// TwinCAT 3 PLC project PLC3
// ProgramVersion: 3.1.4022.3
// libraries:
//   Tc2_Standard, * (Beckhoff Automation GmbH)
//   Tc2_System, * (Beckhoff Automation GmbH)
//   Tc3_Module, * (Beckhoff Automation GmbH)
// project tree:
//   DUTs/ States.TcDUT (not stored)
//   / GlobalTextList.TcGTLO (not stored), PlcTask.TcTTO (not stored), Visualization Manager.TcVMO (not stored)
//   GVLs/ GVL_IO.TcGVL (not stored)
//   POUs/ MAIN.TcPOU, Moving.TcPOU
//   VISUs/ Visualization.TcVIS

// ---- POUs/MAIN.TcPOU
PROGRAM MAIN
VAR
	Timer1 :TON;
	Timer2 : TON;
	PulseTimer1 : TP;

	CurrentState  : States;
	
	ServoRTrigY : R_Trig ; 
	ServoRTrigX : R_Trig ; 
	
	//Eigen trigger booleans
	InitYReady : BOOL;
	InitXReady : BOOL;

	Test : Moving;
	Pos : INT;
	ActualPos : int;
END_VAR

PulseTimer1(IN:=GVL_IO.Start_button, PT:=T#150MS);

Timer1(IN:= GVL_IO.a_1_Vertical_Zaxis_downward, PT:= T#10MS);

CASE CurrentState OF
States.Init:
		//Aanzetten van servo's. Dit kan even duren GEEN HOMING
		GVL_IO.SVONX_SERVO_ON_tableX 	  := TRUE; 
		GVL_IO.SVONY_SERVO_ON_translY 	  := TRUE;
		
		GVL_IO.SETUPX_ORIGIN_tableX := PulseTimer1.Q;
		GVL_IO.SETUPY_ORIGIN_translY := PulseTimer1.Q;
		
		//// Koppelen van outputs Busy aan var's. Triggered op een falling edge.
		IF PulseTimer1.Q THEN
			ServoRTrigX ( clk := gvl_io.SETONX_ORIGIN_tableX ); 
	  		ServoRTrigY ( clk := gvl_io.SETONY_ORIGIN_translationY );
		END_IF
		
		// Bools setten aan de hand van triggers.
		IF ServoRTrigX.Q THEN
			InitXReady:= TRUE;
		END_IF
		
		IF ServoRTrigY.Q THEN
			InitYReady:= TRUE;
		END_IF
		
		// Init voltooid ga naar idle
		IF InitXReady AND InitYReady THEN
			Pos:= 1;
			ActualPos:= 0;
			CurrentState:= States.Idle;
		END_IF
		
States.Idle:
		IF NOT GVL_IO.Stop_button AND NOT GVL_IO.dp2_Cover_detection THEN
			//SEND MESSAGEE TODO
			CurrentState := States.Idle;
		END_IF
		
		IF NOT GVL_IO.Stop_button AND GVL_IO.dp1_Can_detection AND GVL_IO.dp2_Cover_detection THEN
			CurrentState := States.MoveToPickUp; //TODO stopbutton
		END_IF
		
		IF Pos >= 26 THEN
			CurrentState := States.PalletFull;
		END_IF
		
States.MoveToPickUp:

		Test(Position:=0);
		IF NOT Test.Busy THEN
			CurrentState := States.PickUpDown;
		END_IF
		
		
States.PickUpDown:
		IF GVL_IO.a_0_Vertical_Zaxis_upward THEN
			GVL_IO.Aplus_Vert_axis_downwards := TRUE;
		END_IF
		
		IF GVL_IO.a_1_Vertical_Zaxis_downward THEN
			GVL_IO.Vplus_Vacuum_start := TRUE;
			
			IF Timer1.Q THEN
			CurrentState := States.PickUpUp;
			END_IF
		END_IF

States.PickUpUp:
		GVL_IO.Aplus_Vert_axis_downwards := FALSE;
		
		IF GVL_IO.a_0_Vertical_Zaxis_upward THEN
			CurrentState := States.Moving;
		END_IF
		
States.Moving:
		Test(Position:=Pos);
		IF NOT Test.Busy THEN
			Pos:= Pos + 1;
			ActualPos:= ActualPos + 1;
			CurrentState := States.DropDown;
		END_IF
		
States.DropDown:
		IF GVL_IO.a_0_Vertical_Zaxis_upward THEN
			GVL_IO.Aplus_Vert_axis_downwards := TRUE;
		END_IF
		
		IF 	GVL_IO.a_1_Vertical_Zaxis_downward THEN
			GVL_IO.Vplus_Vacuum_start := FALSE;
			Timer2(IN:=GVL_IO.a_1_Vertical_Zaxis_downward, PT:=T#10MS);
			IF Timer2.Q THEN
				CurrentState := States.DropUp;
			END_IF
		END_IF


States.DropUp:
		IF GVL_IO.a_1_Vertical_Zaxis_downward THEN
			GVL_IO.Aplus_Vert_axis_downwards := FALSE;
		END_IF
		
		IF GVL_IO.a_0_Vertical_Zaxis_upward THEN
			CurrentState := States.Idle;
		END_IF
		
States.PalletFull:
		GVL_IO.BR_Alarm_light := TRUE;
		IF GVL_IO.Reset_button THEN
			GVL_IO.BR_Alarm_light := FALSE;
			Pos := 1;
			ActualPos := 0;
			Currentstate := States.Idle;
		END_IF
END_CASE

END_PROGRAM

// ---- POUs/Moving.TcPOU
FUNCTION_BLOCK PUBLIC Moving
VAR_INPUT
	Position : int;
END_VAR
VAR_OUTPUT
END_VAR
VAR
	Busy: BOOL;
	PulseTimer2: TP;
	
	BusyFtrigX : F_Trig;
	BusyFtrigY : F_Trig;
	
	ReadyX : BOOL;
	ReadyY : BOOL;
END_VAR

PulseTimer2(IN:=Busy, PT:=T#150MS);

Busy := TRUE;

CASE Position OF
	0:
		GVL_IO.INX0_from_Input0_tableX := FALSE;
		GVL_IO.INX1_from_Input1_tableX := FALSE;
		GVL_IO.INX2_from_Input2_tableX := TRUE;
		GVL_IO.INY0_from_Input0_translY := TRUE;
		GVL_IO.INY1_from_Input1_translY := FALSE;
		GVL_IO.INY2_from_Input2_translY := TRUE;
	1:
		GVL_IO.INX0_from_Input0_tableX := FALSE;
		GVL_IO.INX1_from_Input1_tableX := FALSE;
		GVL_IO.INX2_from_Input2_tableX := FALSE;
		GVL_IO.INY0_from_Input0_translY := FALSE;
		GVL_IO.INY1_from_Input1_translY := FALSE;
		GVL_IO.INY2_from_Input2_translY := FALSE;
	2:
		GVL_IO.INX0_from_Input0_tableX := TRUE;
		GVL_IO.INX1_from_Input1_tableX := FALSE;
		GVL_IO.INX2_from_Input2_tableX := FALSE;
		GVL_IO.INY0_from_Input0_translY := FALSE;
		GVL_IO.INY1_from_Input1_translY := FALSE;
		GVL_IO.INY2_from_Input2_translY := FALSE;
	3:
		GVL_IO.INX0_from_Input0_tableX := FALSE;
		GVL_IO.INX1_from_Input1_tableX := TRUE;
		GVL_IO.INX2_from_Input2_tableX := FALSE;
		GVL_IO.INY0_from_Input0_translY := FALSE;
		GVL_IO.INY1_from_Input1_translY := FALSE;
		GVL_IO.INY2_from_Input2_translY := FALSE;
	4:
		GVL_IO.INX0_from_Input0_tableX := TRUE;
		GVL_IO.INX1_from_Input1_tableX := TRUE;
		GVL_IO.INX2_from_Input2_tableX := FALSE;
		GVL_IO.INY0_from_Input0_translY := FALSE;
		GVL_IO.INY1_from_Input1_translY := FALSE;
		GVL_IO.INY2_from_Input2_translY := FALSE;
	5:
		GVL_IO.INX0_from_Input0_tableX := FALSE;
		GVL_IO.INX1_from_Input1_tableX := FALSE;
		GVL_IO.INX2_from_Input2_tableX := TRUE;
		GVL_IO.INY0_from_Input0_translY := FALSE;
		GVL_IO.INY1_from_Input1_translY := FALSE;
		GVL_IO.INY2_from_Input2_translY := FALSE;
	6:
		GVL_IO.INX0_from_Input0_tableX := FALSE;
		GVL_IO.INX1_from_Input1_tableX := FALSE;
		GVL_IO.INX2_from_Input2_tableX := FALSE;
		GVL_IO.INY0_from_Input0_translY := TRUE;
		GVL_IO.INY1_from_Input1_translY := FALSE;
		GVL_IO.INY2_from_Input2_translY := FALSE;
	7:
		GVL_IO.INX0_from_Input0_tableX := TRUE;
		GVL_IO.INX1_from_Input1_tableX := FALSE;
		GVL_IO.INX2_from_Input2_tableX := FALSE;
		GVL_IO.INY0_from_Input0_translY := TRUE;
		GVL_IO.INY1_from_Input1_translY := FALSE;
		GVL_IO.INY2_from_Input2_translY := FALSE;
	8:
		GVL_IO.INX0_from_Input0_tableX := FALSE;
		GVL_IO.INX1_from_Input1_tableX := TRUE;
		GVL_IO.INX2_from_Input2_tableX := FALSE;
		GVL_IO.INY0_from_Input0_translY := TRUE;
		GVL_IO.INY1_from_Input1_translY := FALSE;
		GVL_IO.INY2_from_Input2_translY := FALSE;
	9:
		GVL_IO.INX0_from_Input0_tableX := TRUE;
		GVL_IO.INX1_from_Input1_tableX := TRUE;
		GVL_IO.INX2_from_Input2_tableX := FALSE;
		GVL_IO.INY0_from_Input0_translY := TRUE;
		GVL_IO.INY1_from_Input1_translY := FALSE;
		GVL_IO.INY2_from_Input2_translY := FALSE;
	10:
		GVL_IO.INX0_from_Input0_tableX := FALSE;
		GVL_IO.INX1_from_Input1_tableX := FALSE;
		GVL_IO.INX2_from_Input2_tableX := TRUE;
		GVL_IO.INY0_from_Input0_translY := TRUE;
		GVL_IO.INY1_from_Input1_translY := FALSE;
		GVL_IO.INY2_from_Input2_translY := FALSE;
	11:
		GVL_IO.INX0_from_Input0_tableX := FALSE;
		GVL_IO.INX1_from_Input1_tableX := FALSE;
		GVL_IO.INX2_from_Input2_tableX := FALSE;
		GVL_IO.INY0_from_Input0_translY := FALSE;
		GVL_IO.INY1_from_Input1_translY := TRUE;
		GVL_IO.INY2_from_Input2_translY := FALSE;
	12:
		GVL_IO.INX0_from_Input0_tableX := TRUE;
		GVL_IO.INX1_from_Input1_tableX := FALSE;
		GVL_IO.INX2_from_Input2_tableX := FALSE;
		GVL_IO.INY0_from_Input0_translY := FALSE;
		GVL_IO.INY1_from_Input1_translY := TRUE;
		GVL_IO.INY2_from_Input2_translY := FALSE;
	13:
		GVL_IO.INX0_from_Input0_tableX := FALSE;
		GVL_IO.INX1_from_Input1_tableX := TRUE;
		GVL_IO.INX2_from_Input2_tableX := FALSE;
		GVL_IO.INY0_from_Input0_translY := FALSE;
		GVL_IO.INY1_from_Input1_translY := TRUE;
		GVL_IO.INY2_from_Input2_translY := FALSE;
	14:
		GVL_IO.INX0_from_Input0_tableX := TRUE;
		GVL_IO.INX1_from_Input1_tableX := TRUE;
		GVL_IO.INX2_from_Input2_tableX := FALSE;
		GVL_IO.INY0_from_Input0_translY := FALSE;
		GVL_IO.INY1_from_Input1_translY := TRUE;
		GVL_IO.INY2_from_Input2_translY := FALSE;
	15:
		GVL_IO.INX0_from_Input0_tableX := FALSE;
		GVL_IO.INX1_from_Input1_tableX := FALSE;
		GVL_IO.INX2_from_Input2_tableX := TRUE;
		GVL_IO.INY0_from_Input0_translY := FALSE;
		GVL_IO.INY1_from_Input1_translY := TRUE;
		GVL_IO.INY2_from_Input2_translY := FALSE;
	16:
		GVL_IO.INX0_from_Input0_tableX := FALSE;
		GVL_IO.INX1_from_Input1_tableX := FALSE;
		GVL_IO.INX2_from_Input2_tableX := FALSE;
		GVL_IO.INY0_from_Input0_translY := TRUE;
		GVL_IO.INY1_from_Input1_translY := TRUE;
		GVL_IO.INY2_from_Input2_translY := FALSE;
	17:
		GVL_IO.INX0_from_Input0_tableX := TRUE;
		GVL_IO.INX1_from_Input1_tableX := FALSE;
		GVL_IO.INX2_from_Input2_tableX := FALSE;
		GVL_IO.INY0_from_Input0_translY := TRUE;
		GVL_IO.INY1_from_Input1_translY := TRUE;
		GVL_IO.INY2_from_Input2_translY := FALSE;
	18:
		GVL_IO.INX0_from_Input0_tableX := FALSE;
		GVL_IO.INX1_from_Input1_tableX := TRUE;
		GVL_IO.INX2_from_Input2_tableX := FALSE;
		GVL_IO.INY0_from_Input0_translY := TRUE;
		GVL_IO.INY1_from_Input1_translY := TRUE;
		GVL_IO.INY2_from_Input2_translY := FALSE;
	19:
		GVL_IO.INX0_from_Input0_tableX := TRUE;
		GVL_IO.INX1_from_Input1_tableX := TRUE;
		GVL_IO.INX2_from_Input2_tableX := FALSE;
		GVL_IO.INY0_from_Input0_translY := TRUE;
		GVL_IO.INY1_from_Input1_translY := TRUE;
		GVL_IO.INY2_from_Input2_translY := FALSE;
	20:
		GVL_IO.INX0_from_Input0_tableX := FALSE;
		GVL_IO.INX1_from_Input1_tableX := FALSE;
		GVL_IO.INX2_from_Input2_tableX := TRUE;
		GVL_IO.INY0_from_Input0_translY := TRUE;
		GVL_IO.INY1_from_Input1_translY := TRUE;
		GVL_IO.INY2_from_Input2_translY := FALSE;
	21:
		GVL_IO.INX0_from_Input0_tableX := FALSE;
		GVL_IO.INX1_from_Input1_tableX := FALSE;
		GVL_IO.INX2_from_Input2_tableX := FALSE;
		GVL_IO.INY0_from_Input0_translY := FALSE;
		GVL_IO.INY1_from_Input1_translY := FALSE;
		GVL_IO.INY2_from_Input2_translY := TRUE;
	22:
		GVL_IO.INX0_from_Input0_tableX := TRUE;
		GVL_IO.INX1_from_Input1_tableX := FALSE;
		GVL_IO.INX2_from_Input2_tableX := FALSE;
		GVL_IO.INY0_from_Input0_translY := FALSE;
		GVL_IO.INY1_from_Input1_translY := FALSE;
		GVL_IO.INY2_from_Input2_translY := TRUE;
	23:
		GVL_IO.INX0_from_Input0_tableX := FALSE;
		GVL_IO.INX1_from_Input1_tableX := TRUE;
		GVL_IO.INX2_from_Input2_tableX := FALSE;
		GVL_IO.INY0_from_Input0_translY := FALSE;
		GVL_IO.INY1_from_Input1_translY := FALSE;
		GVL_IO.INY2_from_Input2_translY := TRUE;
	24:
		GVL_IO.INX0_from_Input0_tableX := TRUE;
		GVL_IO.INX1_from_Input1_tableX := TRUE;
		GVL_IO.INX2_from_Input2_tableX := FALSE;
		GVL_IO.INY0_from_Input0_translY := FALSE;
		GVL_IO.INY1_from_Input1_translY := FALSE;
		GVL_IO.INY2_from_Input2_translY := TRUE;
	25:
		GVL_IO.INX0_from_Input0_tableX := FALSE;
		GVL_IO.INX1_from_Input1_tableX := FALSE;
		GVL_IO.INX2_from_Input2_tableX := TRUE;
		GVL_IO.INY0_from_Input0_translY := FALSE;
		GVL_IO.INY1_from_Input1_translY := FALSE;
		GVL_IO.INY2_from_Input2_translY := TRUE;
END_CASE

		GVL_IO.DRIVEX_MOVE_tableX := PulseTimer2.Q;
		GVL_IO.DRIVEY_MOVE_translY := PulseTimer2.Q;
		
		//// Koppelen van outputs Busy aan var's. Triggered op een falling edge.
	   	BusyFtrigX ( clk := gvl_io.BUSYX_BUSY_tableX ); 
	  	BusyFtrigY ( clk := gvl_io.BUSYY_BUSY_traslationY );
		
		// Bools setten aan de hand van triggers.
		IF BusyFtrigX.Q THEN
			ReadyX:= TRUE;
		END_IF
		
		IF BusyFtrigY.Q THEN
			ReadyY:= TRUE;
		END_IF
		
		// Init voltooid ga naar idle
		IF ReadyY AND ReadyX THEN
			GVL_IO.DRIVEX_MOVE_tableX := FALSE;
			GVL_IO.DRIVEY_MOVE_translY := FALSE;
			ReadyX:= FALSE;
			ReadyY:= FALSE;
			Busy:= FALSE;
			//CurrentState := States.PickUpDown;
		END_IF

END_FUNCTION_BLOCK

// ---- VISUs/Visualization.TcVIS
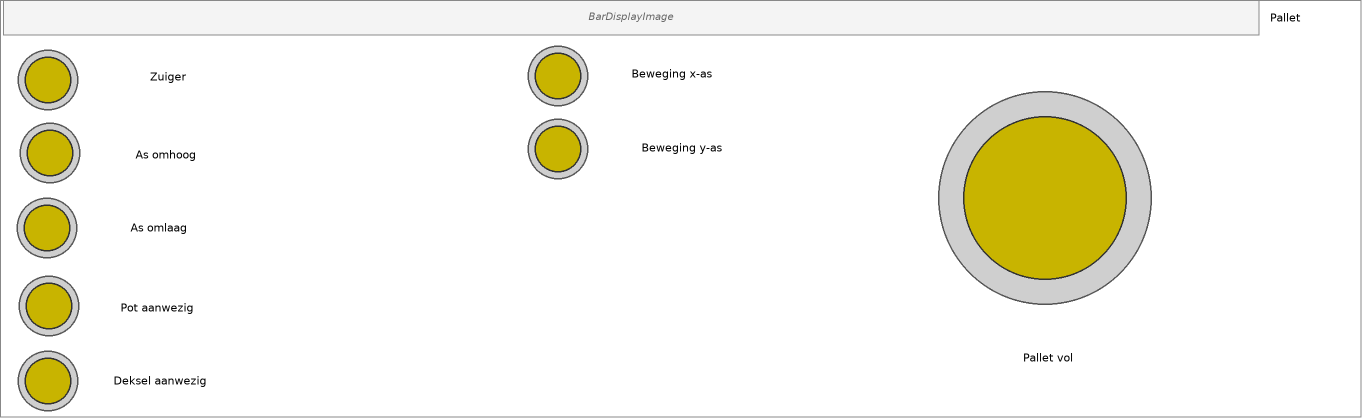
VISUALIZATION Visualization  // 1362x418
    Label (1211,3 149x30), "Pallet"
    Lamp1 (13,45 70x70), variable: GVL_IO.Vplus_Vacuum_start, style: Lamp-Lamp1-Yellow
    Label (93,62 150x30), "Zuiger"
    Lamp1 (15,118 70x70), variable: GVL_IO.a_0_Vertical_Zaxis_upward, style: Lamp-Lamp1-Yellow
    Label (91,140 150x30), "As omhoog"
    Lamp1 (12,193 70x70), variable: GVL_IO.a_1_Vertical_Zaxis_downward, style: Lamp-Lamp1-Yellow
    Label (84,213 150x30), "As omlaag"
    Lamp1 (14,271 70x70), variable: GVL_IO.dp1_Can_detection, style: Lamp-Lamp1-Yellow
    Label (82,293 150x30), "Pot aanwezig"
    Lamp1 (13,346 70x70), variable: GVL_IO.dp2_Cover_detection, style: Lamp-Lamp1-Yellow
    Label (85,366 150x30), "Deksel aanwezig"
    Lamp1 (523,41 70x70), variable: GVL_IO.BUSYX_BUSY_tableX, style: Lamp-Lamp1-Yellow
    Label (597,59 150x30), "Beweging x-as"
    Lamp1 (523,114 70x70), variable: GVL_IO.BUSYY_BUSY_traslationY, style: Lamp-Lamp1-Yellow
    Label (607,133 150x30), "Beweging y-as"
    Lamp1 (921,67 248x262), variable: GVL_IO.BR_Alarm_light, style: Lamp-Lamp1-Yellow
    Label (973,343 150x30), "Pallet vol"
    BarDisplayImage (3,-2 1256x37), value: MAIN.ActualPos, style: BarDisplayImage-Gray, scale format: %.1f, scale 0..25
END_VISUALIZATION
